{attribute 'qualified_only'}
VAR_GLOBAL CONSTANT
	// Encoder reference values in counts = nm
	// Put encoder reference values for nominal 0 here
	nM2K2X_ENC_REF : ULINT := 6077000; //these numbers
	nM2K2Y_ENC_REF : ULINT := 5975460; //are
	nM2K2rX_ENC_REF : ULINT := 50412360;//real
END_VAR

(* stored: Version 1.1.0.1, ProductVersion 3.1.4022.18
   GVL GVL_M2K2: Id {b80c1e96-150a-4c40-81ca-c5a63f5628f5} *)
